// TIA Portal V20 export
// export: Created 2025-12-01T14:57:16.5185292Z, ExportSetting None, DisplayName Totally Integrated Automation Portal, DisplayVersion V20 Update 3, DisplayName TIA Portal Openness, DisplayVersion V20 Update 3, DisplayName TIA Portal Version Control Interface, DisplayVersion V20 Update 3, DisplayName STEP 7 Professional, DisplayVersion V20 Update 3, DisplayName STEP 7 Safety, DisplayVersion V20 Update 2, DisplayName WinCC Basic/Comfort/Advanced, DisplayVersion V20 Update 3, DisplayName WinCC Professional, DisplayVersion V20 Update 3, DisplayName WinCC Unified, DisplayVersion V20 Update 3
DATA_BLOCK "DB900_Estado_Mesas"   // DB900
{ S7_Optimized_Access := 'FALSE' }
AUTHOR : GENERAL
NAME : 20160413
VERSION : 3.1
// stored: AutoNumber false
   VAR RETAIN
      EstadoVI { S7_SetPoint := 'True'} : Array[0.."CTE_MaxMesas"] of "EstadosMesa";
      MoviManual { S7_SetPoint := 'True'} : Array[0.."CTE_MaxMesas"] of "MoviManualMesa";
   END_VAR
BEGIN
END_DATA_BLOCK
